(* PLC project ComparisonTest *)
(* stored: creationDateTime 2024-01-01T00:00:00, modificationDateTime 2024-01-01T00:00:00 *)

PROGRAM Main
  VAR
    X001 : BOOL;
    TempSensor : INT;
    Threshold : INT;
    Y001 : BOOL;
    Y002 : BOOL;
    SumResult : INT;
  END_VAR
  VAR  (* added by the conversion: wires and edge detectors of the diagram *)
    _EQ10_OUT : BOOL;
  END_VAR

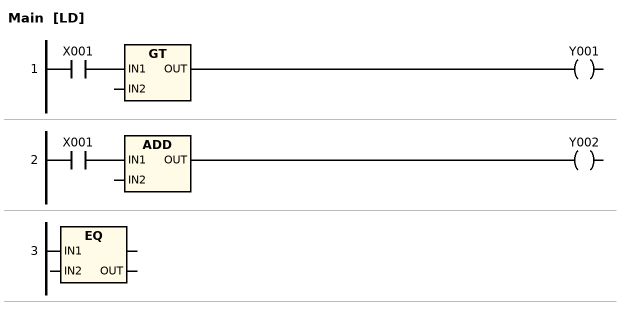
(* LD diagram, written out as Structured Text *)
Y001 := GT(IN1 := X001);
Y002 := ADD(IN1 := X001);
_EQ10_OUT := EQ(IN1 := TRUE);
END_PROGRAM

CONFIGURATION Config
  RESOURCE Res ON PLC
    TASK Main(INTERVAL := T#20ms, PRIORITY := 0);
    PROGRAM Main WITH Main : Main;
  END_RESOURCE
END_CONFIGURATION
